TYPE I64 : LINT; END_TYPE

(* stored: Version 1.1.0.1
   DUT I64: Id {08127285-333f-0c28-05c5-230d42ceb5be} *)
